(* CoDeSys 2.3.9.37 project: Cap12_8.pro *)
(* Libraries: Util.lib 18.5.10 16:14:28, Standard.lib 4.10.05 12:14:46, IecSfc.lib 13.4.06 16:51:28 *)

(* Global variable list: Global_Variables *)
VAR_GLOBAL
   (* Entradas PLC *)
   IW1_Posicion : WORD;   (* Posición real de la valvula *)
   IX2_Error : BOOL;         (* Error en la Válvula *)
    IW2_Caudal : WORD;  (*Lectura del caudalímetro *)

   (* Variables para el control de la visualización *)
   (*Panel de control de la valvula 1 *)
   Man : BOOL;  (* Manual/Automarico *)
   RefManual : REAL;  (* SP Manual en lazo abierto*)
   (* Panel de control del controlador PI *)
   ManPI : BOOL;  (* Manual/Automatico PI *)
   ManPI_Ent: REAL;  (* Valor de entrada del PI Manual *)
   KpPI : REAL := 0.2; (*Parametro Kp del PI *)
   TNPI:REAL := 400;  (* Tiempo Integral del PI *)
  SPPI:REAL := 30;  (* Set Point del PI en modo lazo cerrado *)



   (*Salidas *)
   QW1_SPPosicion : WORD;  (* Consigna de posición para la válvula *)


(*-----------------------------------------------------*)

(* Otras variables  de la simulación*)
   QX3_ValvulaONOFF: BOOL; (* Apertura cierre válvula ON/OFF *)



END_VAR

(* POU PLC_PRG, ST *)
PROGRAM PLC_PRG
VAR
END_VAR
 Proceso();
 ProgramaControl();
END_PROGRAM

(* POU Proceso, ST *)
PROGRAM Proceso
VAR
       (* Parámetros del sistema posición válvula *)
       K: REAL :=1;
       tau : REAL:=500;
       (* Parámetros del sistema Posición-Caudal *)
       K1: REAL :=0.6;
       tau1 : REAL:=3000;
      (* Variables de tiempo *)
	tact: TIME;
	tactw: DWORD;
	tinc: REAL;
	toldw: DWORD;
      (* Variables del Proceso *)
      Pos : REAL;
     SP_Pos:REAL;
     Caudal:REAL;
      Ciclo1:BOOL:=TRUE;
	EscalaSalida: Escalado;
	IW1R: REAL;
      IW2R:REAL;
	EscalaEntrada: Escalado;
	QW1R: REAL;
	EscalaPos: Escalado;
	EscalaCaudal: Escalado;
END_VAR
  (* Lectura de la consigna de la posición y paso a real *)
  QW1R:=WORD_TO_REAL(QW1_SPPosicion);
  EscalaEntrada(Valor_Ent:=QW1R,Min_Ent:=0,Max_Ent:=4095,Min_Sal:=0,Max_Sal:=100,Valor_Sal=>SP_Pos);

    (* Programa que simula un sistema de primer orden *)
    tact:=TIME();
    tactw:=TIME_TO_DWORD(tact);
    (* Calcula el intervalo de tiempo desde el último ciclo en milisegundos *)
    tinc:=DWORD_TO_REAL(tactw-toldw);
    (* Almacena el valor actual para al próximo ciclo *)
    toldw:=tactw;



    IF Ciclo1=FALSE THEN
        Pos:=Pos+tinc*(K*SP_Pos-Pos)/tau;
        Caudal:=Caudal+tinc*(K1*Pos-Caudal)/tau1;
    ELSE
        Ciclo1:=FALSE;
    END_IF

    EscalaPos(Valor_Ent:=Pos,Min_Ent:=0,Max_Ent:=100,Min_Sal:=0,Max_Sal:=4095,Valor_Sal=>IW1R);
    IW1_Posicion:=REAL_TO_WORD(IW1R);
     EscalaCaudal(Valor_Ent:=Caudal,Min_Ent:=0,Max_Ent:=100,Min_Sal:=0,Max_Sal:=4095,Valor_Sal=>IW2R);
    IW2_Caudal:=REAL_TO_WORD(IW2R);
END_PROGRAM

(* POU Escalado, ST *)
FUNCTION_BLOCK Escalado
VAR_INPUT
	Valor_Ent : REAL;    (* Valor a convertir *)
	Min_Ent : REAL;      (* Valor mínimo de la entrada *)
	Max_Ent : REAL;	  (* Valor máximo de la entrada *)
	Min_Sal : REAL;      (* Valor mínimo de la salida *)
	Max_Sal : REAL;	   (* . Valor máximo de la salida. *)
       ValError : REAL:=-1;    (*Valor al que poner la salida en caso de error *)
END_VAR
VAR_OUTPUT
	Valor_Sal : REAL;   (*. Valor convertido *)
	Error :  BOOL;         (* Se activa cuando el valor de entrada queda fuera de límites *)
END_VAR
VAR
	pendiente: REAL;
END_VAR
Error:= (Valor_Ent>Max_Ent) OR (Valor_Ent<Min_Ent);

IF NOT Error THEN
   pendiente:=(Max_Sal-Min_Sal)/(Max_Ent-Min_Ent);
   Valor_Sal:=Valor_Ent*pendiente+Min_Sal;
ELSE
   Valor_Sal:=ValError;
END_IF
END_FUNCTION_BLOCK

(* POU ControladorPI, ST *)
FUNCTION_BLOCK ControladorPI
VAR_INPUT
	Y :REAL;       (* Variable a controlar. *)
	SP : REAL;    (* Set Point, valor deseado de la variable a controlar.*)
	Kp : REAL := 1;     (* Parámetro del controlador. Proporcionar un valor por defecto de 1.0.*)
       TN : REAL:=1;       (* Parámetro del controlador *)
	Umin  : REAL :=0;   (* Valor mínimo de la salida. Por defecto tendrá el valor 0 *)
	UMax : REAL:=100;   (* Valor máximo de la salida. Por defecto, tendrá un valor 100.0.*)
	Offset :REAL:=0;     (* Cantidad a sumar a la señal del controlador. Por defecto tendrá un valor 0.*)
	Manual : BOOL;      (* TRUE modo manual, FALSE modo automático*)
	Manual_Ent : REAL;   (*Valor para la salida según ecuación (1.3) en modo manual *)
END_VAR
VAR_OUTPUT
	U : REAL;    (*Salida del controlador. *)
      Lim : BOOL;  (*Estará a TRUE si se superan los límites Umin o Umax en la salida *)
END_VAR
VAR
	tact: TIME;
	tactw: DWORD;
	tinc: REAL;
	toldw: DWORD;
	error: REAL;
	ierror: REAL;
      Ciclo1:BOOL :=TRUE;
END_VAR
   (* Calcula el instante de tiempo actual y se pasa a DWORD en milisegundos *)
    tact:=TIME();
    tactw:=TIME_TO_DWORD(tact);
    (* Calcula el intervalo de tiempo desde el último ciclo en milisegundos *)
    tinc:=DWORD_TO_REAL(tactw-toldw);
    (* Almacena el valor actual para al próximo ciclo *)
    toldw:=tactw;

IF Manual THEN
   U:=Manual_Ent+Offset;
   ierror:=0;
ELSE

    (* Calculo error ¨*)
   error:=SP-Y;
   (* Calculo de la integral del error  usando el método de Euler*)
   IF NOT Ciclo1 THEN
       ierror:=ierror+tinc*error;
  END_IF

   (* Calculo de la salida del conttrolador *)
  U:=Kp*(error+(1/TN)*ierror)+Offset;


END_IF


IF Ciclo1 THEN
   U:=Offset;
   Ciclo1:=FALSE;
END_IF


IF U>Umax THEN
     U:=Umax;
ELSE
   IF U<Umin THEN
       U:=Umin;
   END_IF
END_IF

LIM:=(U>Umax) OR  (U<Umin);
END_FUNCTION_BLOCK

(* POU ControlValvula, ST *)
FUNCTION_BLOCK ControlValvula
VAR_INPUT
    Manual : BOOL;
    SPManual : REAL;
    SPAuto : REAL;
    PV : REAL;
    ErrorValvula : BOOL;
    SPError : REAL;
     Encl : BOOL;
     SPEncl : REAL;
END_VAR
VAR_OUTPUT
      SP:REAL;
      DIF : REAL;
      Alarma : BOOL;
END_VAR
VAR
	TempoError: TON;
	INTempo: BOOL;
END_VAR
IF MANUAL THEN
     SP:=SPManual;
ELSE
     SP:= SPAuto;
END_IF

(* Se le da prioridad al enclavamiento *)
IF Encl THEN SP:=SPEncl;  END_IF

DIF:=SP-PV;
INTempo:= ABS(DIF)>0.3;
TempoError(IN:=INTempo, PT:=T#10h);

Alarma:=ErrorValvula OR TempoError.Q;
(* Prioridad máxima a la salida de error *)
IF (Alarma) THEN  SP:=SPError;   END_IF
END_FUNCTION_BLOCK

(* Visualisation Visu
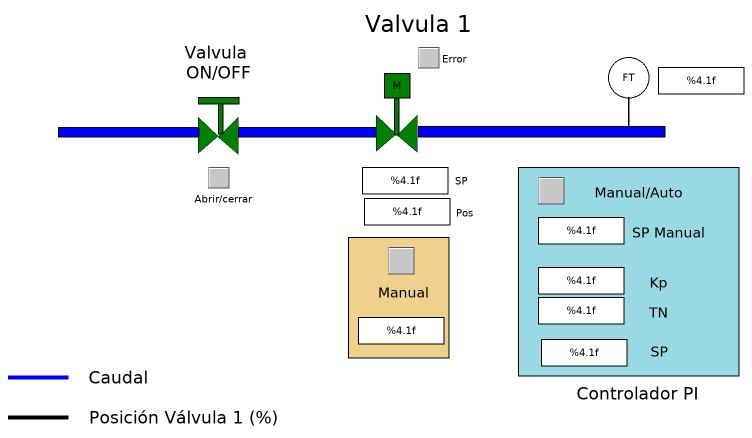
button at (490,260)-(516,287): toggles Man
rectangle at (460,330)-(546,357): text "%4.1f"; shows RefManual; editable 0..100
polygon at (478,128)-(499,164): alarm colour if IX2_Error
polygon at (499,128)-(519,165): alarm colour if IX2_Error
rectangle at (486,86)-(512,111): text "M"; alarm colour if IX2_Error
rectangle at (496,111)-(501,148): alarm colour if IX2_Error
rectangle at (464,180)-(550,207): text "%4.1f"; shows Proceso.SP_Pos
rectangle at (547,182)-(580,206): text "SP"
rectangle at (550,214)-(583,238): text "Pos"
rectangle at (480,290)-(531,321): text "Manual"
rectangle at (466,211)-(552,238): text "%4.1f"; shows Proceso.Pos
button at (520,60)-(541,81): toggles IX2_Error
rectangle at (540,60)-(573,84): text "Error"
rectangle at (460,20)-(581,54): text "Valvula 1"
polygon at (320,130)-(340,167): alarm colour if QX3_ValvulaONOFF
polygon at (300,130)-(321,166): alarm colour if QX3_ValvulaONOFF
rectangle at (320,110)-(325,147): alarm colour if QX3_ValvulaONOFF
rectangle at (300,110)-(341,117): alarm colour if QX3_ValvulaONOFF
rectangle at (260,50)-(381,101): text "Valvula / ON/OFF"
button at (310,180)-(331,201): toggles QX3_ValvulaONOFF
rectangle at (290,200)-(361,224): text "Abrir/cerrar"
rectangle at (140,370)-(301,411): text "Caudal"
ellipse at (710,70)-(751,111): text "FT"
button at (640,190)-(666,217): toggles ManPI
rectangle at (659,386)-(820,427): text "Controlador PI"
rectangle at (680,190)-(801,221): text "Manual/Auto"
rectangle at (710,230)-(831,261): text "SP Manual"
rectangle at (640,230)-(726,257): text "%4.1f"; shows ManPI_Ent; editable 0..100
rectangle at (640,280)-(726,307): text "%4.1f"; shows KpPI; editable 0..100
rectangle at (640,310)-(726,337): text "%4.1f"; shows TNPI; editable 0..1000
rectangle at (720,280)-(801,311): text "Kp"
rectangle at (720,310)-(801,341): text "TN"
rectangle at (760,80)-(846,107): text "%4.1f"; shows Proceso.Caudal
rectangle at (643,352)-(729,379): text "%4.1f"; shows SPPI; editable 0..100
rectangle at (721,349)-(802,380): text "SP"
rectangle at (140,410)-(431,451): text "Posición Válvula 1 (%)"
8 more shapes without text or variables
1 elements of other kinds (tables, trends, ...) not read
*)
